(* IEC 61131-3 sources: CannyIEC/extracted_st/cannyiec/globalvariables/variables, 1 file *)

(* ---- Variables.st ---- *)
(* --- Interface --- *)
{attribute 'qualified_only'}
//{attribute 'conditionalshow'}
//{attribute 'conditionalshow' := 'SomeText'}
//{attribute 'hide'}
VAR_GLOBAL
    g_iDummy : INT; /// This is a dummy global variable
END_VAR
